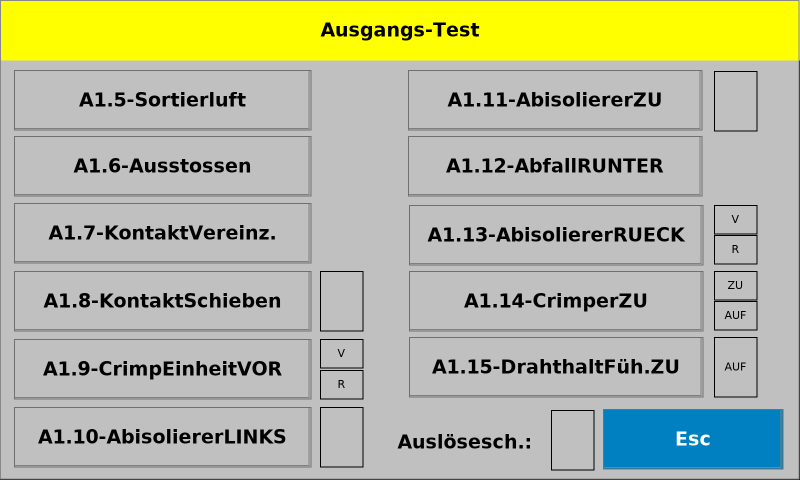
VISUALIZATION OutTest  // 800x480
    Rectangle (0,0 800x480)
    Rectangle (0,0 800x60), "Ausgangs-Test"
    Button (603,409 180x60), "Esc"
        OnMouseUp: change screen: Previous Start
        OnMouseUp: execute { P_SaveCurrentLanguage(); }
    Button (14,70 297x60), "A1.5-Sortierluft", colour toggle: DB6.frceY11SortierLuft
        toggle DB6.frceY11SortierLuft
    Button (14,136 297x60), "A1.6-Ausstossen", colour toggle: DB6.frceY1Ausstossen
        toggle DB6.frceY1Ausstossen
    Button (14,203 297x60), "A1.7-KontaktVereinz.", colour toggle: DB6.frceY2KontaktVereinzelung
        toggle DB6.frceY2KontaktVereinzelung
    Button (14,339 297x60), "A1.9-CrimpEinheitVOR", colour toggle: DB6.frceY4CrimpEinheitVOR
        toggle DB6.frceY4CrimpEinheitVOR
    Button (14,407 297x60), "A1.10-AbisoliererLINKS", colour toggle: DB6.frceY5AbisolierNachLINKS
        toggle DB6.frceY5AbisolierNachLINKS
    Button (14,271 297x60), "A1.8-KontaktSchieben", colour toggle: DB6.frceY3KontaktSchieben
        toggle DB6.frceY3KontaktSchieben
    Button (408,70 294x60), "A1.11-AbisoliererZU", colour toggle: DB6.frceY6AbisoliererZU
        toggle DB6.frceY6AbisoliererZU
    Button (409,205 294x60), "A1.13-AbisoliererRUECK", colour toggle: DB6.frceY8AbisoliererRUECK
        toggle DB6.frceY8AbisoliererRUECK
    Button (409,271 294x60), "A1.14-CrimperZU", colour toggle: DB6.frceY9CrimperZU
        toggle DB6.frceY9CrimperZU
    Button (409,337 294x60), "A1.15-DrahthaltFüh.ZU", colour toggle: DB6.frceY10DrahthaltFuehrungZU
        toggle DB6.frceY10DrahthaltFuehrungZU
    Button (408,136 294x60), "A1.12-AbfallRUNTER", colour toggle: DB6.frceY7AbfallRUNTER
        toggle DB6.frceY7AbfallRUNTER
    Rectangle (320,271 43x60), colour toggle: IO.inKontaktSchiebenVORN
    Rectangle (320,339 43x29), "V", colour toggle: IO.inCrimpEinheitIstVORN
    Rectangle (320,370 43x29), "R", colour toggle: IO.inCrimpEinheitIstRUECK
    Rectangle (320,407 43x60), colour toggle: IO.inAbisoliererIstLINKS
    Rectangle (714,301 43x29), "AUF", colour toggle: IO.inCrimpZangeIstOFFEN
    Rectangle (714,271 43x29), "ZU", colour toggle: IO.inCrimpZangeIstZU
    Rectangle (714,235 43x29), "R", colour toggle: IO.inAbisoliererIstRUECK
    Rectangle (714,205 43x29), "V", colour toggle: IO.inAbisoliererIstVORN
    Rectangle (714,71 43x60), colour toggle: IO.inAbisoliererIstZU
    Rectangle (714,337 43x60), "AUF", colour toggle: IO.inDrahthalterIstOffen
    Rectangle (551,410 43x60), colour toggle: IO.inAusloeseSchalter
    Label (388,427 154x30), "Auslösesch.:"
END_VISUALIZATION

(* stored: Version 1.1.0.1, ProductVersion 3.1.4024.3
   Visu OutTest: Id {9834cd0f-ff1d-4e80-ae88-424c36b51648} *)
